// TIA Portal V17 export
// export: Created 2023-12-05T13:40:23.2087961Z, ExportSetting WithDefaults, DisplayName Totally Integrated Automation Portal, DisplayVersion V17, DisplayName TIA Portal Openness, DisplayVersion V17, DisplayName TIA Portal Version Control Interface, DisplayVersion V17, DisplayName SINAMICS Startdrive Advanced, DisplayVersion V17, DisplayName SINAMICS Startdrive G130, G150, S120, S150, SINAMICS MV, S210, DisplayVersion V17, DisplayName SINAMICS Startdrive G110M, G120, G120C, G120D, G120P, G115D, DisplayVersion V17, DisplayName STEP 7 Professional, DisplayVersion V17, DisplayName STEP 7 Safety, DisplayVersion V17, DisplayName WinCC Professional, DisplayVersion V17
FUNCTION "FC534 FSU_V5_1_7 Alarms" : Void   // FC534, LAD
{ S7_Optimized_Access := 'TRUE' }
VERSION : 0.1
// LG 30.06.2022 => Changed name of the block (structures are the same like in STD Block V5.1.6
// 10.06.2020 => created for V5_1_0 SB
// 08.09.2021 => Changed name of the block (structures are the same like in STD Block V 5_1_0)
// stored: AutoNumber false, IsIECCheckEnabled false, SetENOAutomatically false, UDAEnableTagReadback false
   VAR_INPUT
      AckStep : Bool;
      "SB DB" : Int;
      "Alarm DB" : Int;
      "Alarm Offset" : Int;
   END_VAR
   VAR_TEMP
      "SB DBW" : Word;
      "AL DBW" : Word;
      "TR DBW" : Word;
   END_VAR
BEGIN

NETWORK
TITLE = Initialization
      L     #"SB DB";
      T     #"SB DBW";
      L     #"Alarm DB";
      T     #"AL DBW";
      L     #"Alarm Offset";
      SLD   3;
      LAR1;

NETWORK
TITLE = Cylinder faults
      CLR;
      OPN   DB [#"SB DBW"];
      L     %DBW70;
      OPN   DB [#"AL DBW"];
      T     DBW [AR1, P#0.0];

NETWORK
TITLE = RCFaults
      A     #AckStep;
      JCN   eno;
      CLR;
      OPN   DB [#"SB DBW"];
      L     %DBB74;
      OPN   DB [#"AL DBW"];
      T     DBB [AR1, P#2.0];
eno:  NOP   0;

NETWORK
TITLE = Faults
      CLR;
      OPN   DB [#"SB DBW"];
      L     %DBB76;
      OPN   DB [#"AL DBW"];
      T     DBB [AR1, P#4.0];
END_FUNCTION
